% RSLogix 500 project PI_EnfoqueContinuo.RSS, saved by version 8.30.00.15 %
PROJECT "UNTITLED"    % processor: Bul.1763 MicroLogix 1100 Series B %

PROGRAM FILES
  LAD 2   13 rungs

DATA FILES
  O0 OUTPUT  6 elements
  I1 INPUT  12 elements
  S2 STATUS  66 elements
  B3 BINARY  1 elements
  T4 TIMER  1 elements
  C5 COUNTER  1 elements
  R6 CONTROL  1 elements
  N7 INTEGER  12 elements
  F8 FLOAT  9 elements
  PD9   1 elements

LADDER 2
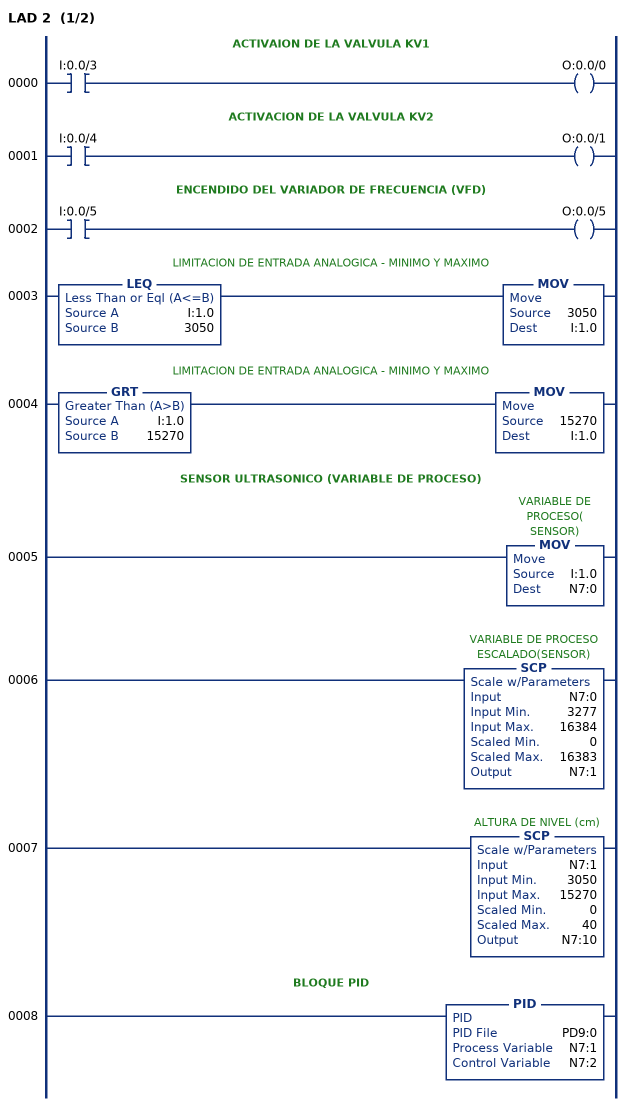
% Rung: 0 %
% TITLE: ACTIVAION DE LA VALVULA KV1 %
SOR XIC I:0.0/3 OTE O:0.0/0 EOR
% Rung: 1 %
% TITLE: ACTIVACION DE LA VALVULA KV2 %
SOR XIC I:0.0/4 OTE O:0.0/1 EOR
% Rung: 2 %
% TITLE: ENCENDIDO DEL VARIADOR DE FRECUENCIA (VFD) %
SOR XIC I:0.0/5 OTE O:0.0/5 EOR
% Rung: 3 %
% LIMITACION DE ENTRADA ANALOGICA - MINIMO Y MAXIMO %
SOR LEQ I:1.0 3050 MOV 3050 I:1.0 EOR
% Rung: 4 %
% LIMITACION DE ENTRADA ANALOGICA - MINIMO Y MAXIMO %
SOR GRT I:1.0 15270 MOV 15270 I:1.0 EOR
% Rung: 5 %
% TITLE: SENSOR ULTRASONICO (VARIABLE DE PROCESO) %
SOR MOV I:1.0 N7:0 EOR
%   N7:0  "VARIABLE DE PROCESO(SENSOR)" %
% Rung: 6 %
SOR SCP N7:0 3277 16384 0 16383 N7:1 EOR
%   N7:0  "VARIABLE DE PROCESO(SENSOR)" %
%   N7:1  "VARIABLE DE PROCESO ESCALADO(SENSOR)" %
% Rung: 7 %
SOR SCP N7:1 3050 15270 0 40 N7:10 EOR
%   N7:1  "VARIABLE DE PROCESO ESCALADO(SENSOR)" %
%   N7:10  "ALTURA DE NIVEL (cm)" %
% Rung: 8 %
% TITLE: BLOQUE PID %
SOR PID PD9:0 N7:1 N7:2 EOR
%   N7:1  "VARIABLE DE PROCESO ESCALADO(SENSOR)" %
%   N7:2  "VARIABLE DE CONTROL (PID)" %

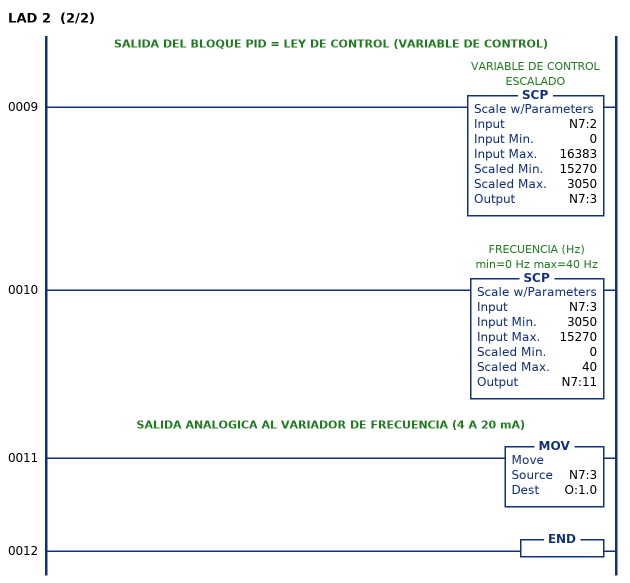
% Rung: 9 %
% TITLE: SALIDA DEL BLOQUE PID = LEY DE CONTROL (VARIABLE DE CONTROL) %
SOR SCP N7:2 0 16383 15270 3050 N7:3 EOR
%   N7:2  "VARIABLE DE CONTROL (PID)" %
%   N7:3  "VARIABLE DE CONTROL ESCALADO" %
% Rung: 10 %
SOR SCP N7:3 3050 15270 0 40 N7:11 EOR
%   N7:3  "VARIABLE DE CONTROL ESCALADO" %
%   N7:11  "FRECUENCIA (Hz) min=0 Hz max=40 Hz" %
% Rung: 11 %
% TITLE: SALIDA ANALOGICA AL VARIADOR DE FRECUENCIA (4 A 20 mA) %
SOR MOV N7:3 O:1.0 EOR
%   N7:3  "VARIABLE DE CONTROL ESCALADO" %
% Rung: 12 %
SOR END EOR

DATA TABLE (non-zero values as saved)
DATA B3
% B3:0 % 0X0001
DATA N7
% N7:0 % 8364 6358 10297 7590 6270 0 0 0 0 0
% N7:10 % 11 15
DATA F8
% F8:0 % 3 200 0.7003891 0.003356934 16384
